// Mitsubishi GX Works2 project: 실린더 제어 예제 1   PLC: Q03UDV

PROGRAM MAIN
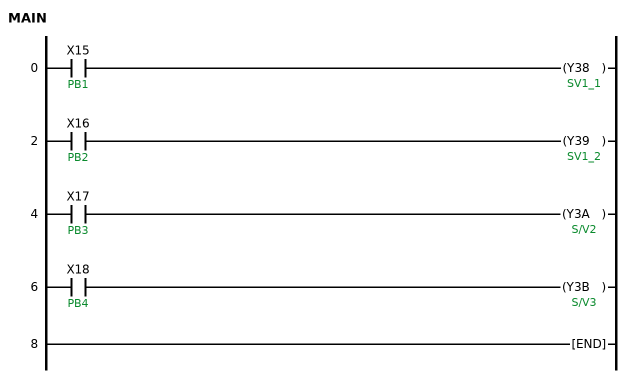
0     LD      X15  ; PB1
      OUT     Y38  ; SV1_1
2     LD      X16  ; PB2
      OUT     Y39  ; SV1_2
4     LD      X17  ; PB3
      OUT     Y3A  ; S/V2
6     LD      X18  ; PB4
      OUT     Y3B  ; S/V3
8     END
END_PROGRAM
